{attribute 'GeneratedUsingTerminal: EJ2502-0000-0023'}
{attribute addProperty BoxType "EJ2502-0000-0023"}
{attribute addProperty Id "PWM_outputAT %Q*UINT2"}
{attribute addProperty CRC "1281526221"}
{attribute addProperty Size "2"}
TYPE PWM_Outputs_Channel_4C6289CD EXTENDS OutputBase_10CEE7DE :
STRUCT
	{attribute addProperty Name "PWM_output"}
	PWM_output AT %Q* : UINT;
END_STRUCT
END_TYPE

(* stored: Version 1.2.0.0, ProductVersion 3.1.4024.11
   DUT PWM_Outputs_Channel_4C6289CD: Id {3ee0c9bd-336b-4f01-8a7f-e33571e33093} *)
